(* Logix 5000 project; controller DC01 vendor 1 type 14 code 165 rev 32.12; software revision 32.04; part 2 of 13 *)
(* tags used below, declared in another part *)
   LN01_Main_Messages : DINT[250];
   LN01_Schedule : UDT_Current_Status;
   LN01_ScheduleUnits_Produced_from_line : DINT;
   LN01_Weekly_Schedule : UDT_Weekly_Schedule;

PROGRAM LN01   (* main routine MainRoutine *)
VAR
   Always_Off : BOOL;
   Average_Array : DINT[20] := ([0] := 1, [2] := 1, [8] := 1, [9] := 1);
   Average_Sum : DINT := 4;
   Averaged_LineSpeed : REAL := 0.0004;
   badModel : STRING_40;
   BlockStarveLocal : DINT;
   Break1_Hour : DINT;
   Break1_Hour_String : STRING;
   Break1_Length : DINT;
   Break1_MilliRemain : DINT;
   Break1_Min : DINT;
   Break1_Min_String : STRING;
   Break1_MinDisplay : DINT;
   Break1_SecDisplay : DINT;
   Break1_SecRemain : DINT;
   Break1_SecWholeMin : DINT;
   Break1_Timer : TIMER;
   Break2_Hour : DINT;
   Break2_Hour_String : STRING;
   Break2_Length : DINT;
   Break2_MilliRemain : DINT;
   Break2_Min : DINT;
   Break2_Min_String : STRING;
   Break2_MinDisplay : DINT;
   Break2_SecDisplay : DINT;
   Break2_SecRemain : DINT;
   Break2_SecWholeMin : DINT;
   Break2_Timer : TIMER;
   Break_1stStation : BOOL;
   Break_LineWide : BOOL;
   Break_WorkCenter : BOOL;
   Break_Workstation : BOOL;
   dlw_test : DINT := -805278210;
   End_Hour : DINT := 20;
   End_Hour_String : STRING := '20';
   End_Min : DINT := 3;
   End_Min_String : STRING := '3-';
   faultcount : DINT;
   FaultExists : CONTROL := (LEN := 230);
   firstCharacter : STRING_40 := 'W';
   FlexTimer_HoursDisplay : DINT;
   FlexTimer_MinutesDisplay : DINT;
   FlexTimer_SecondsDisplay : DINT;
   FlexTimertoHours : DINT;
   FlexTimertoMinutes : DINT;
   FlexTimertoSeconds : DINT;
   HoursFromMidnight : DINT;
   HoursFromMidnight_Remain : DINT;
   HoursTilMidnight : DINT;
   HoursTilMidnight_Remain : DINT;
   KnownFaultExist : DINT := 5;
   L02EAS35 : DINT;
   L02EDM16 : DINT;
   LineRate_perSecond_scheduled : DINT;
   LN01_Flex_Timer : TIMER;
   LN01_MachineOverAll_MNTa : DINT;
   LN01_MainLine_MSG : MESSAGE;
        MessageParameters(ServiceCode := 16#004c, LocalElement := LN01_Main_Messages[0], ...)
   LN01_ML_Message_MSG : MESSAGE;
   LN01_Rotate_Timer : TIMER;
   LN01_SNModel_MSG : MESSAGE;
   LN02EAS35 : DINT;
   LN02EDM16 : DINT;
   Local_Counter : COUNTER[20] := ([0].PRE := 1);
   Local_DATETIME : DINT[20];
   Local_Timer : TIMER[30] := ([0].EN := 1, [0].DN := 1, [3].PRE := 1000, [3].ACC := 429, [3].EN := 1, [3].TT := 1, [4].PRE := 400, [4].ACC := 272, [4].EN := 1, [4].TT := 1, [6].PRE := 2000, [6].ACC := 194, [6].EN := 1, [6].TT := 1);
   local_timer2 : TIMER := (PRE := 1000, ACC := 629, EN := 1, TT := 1);
   Lunch_Hour : DINT;
   Lunch_Hour_String : STRING;
   Lunch_Length : DINT;
   Lunch_MilliRemain : DINT;
   Lunch_Min : DINT;
   Lunch_Min_String : STRING;
   Lunch_MinDisplay : DINT;
   Lunch_SecDisplay : DINT;
   Lunch_SecRemain : DINT;
   Lunch_SecWholeMin : DINT;
   Lunch_Timer : TIMER;
   Midnight_Hour : DINT;
   mlc_test21 : BOOL;
   null : STRING;
   OneShot : DINT;
   ONS_0 : DINT := 536870912;
   ONS_20 : DINT;
   prevCalculateLocal : DINT;
   PreviousCount : DINT := 554;
   previousSerialNumber : STRING := 'CA0807422';
   PreviousShift : DINT := 1;
   readIndex : DINT := 41;
   register : DINT := 5;
   Rotate_MilliRemain : DINT;
   Rotate_Seconds_perShift : DINT;
   Rotate_SecRemain : DINT;
   RTO_Test : TIMER := (PRE := 2000, ACC := 2000, DN := 1);
   Scheduled_Units_Buffer : DINT := 1240;
   Shift_Break_Lengths : DINT;
   Shift_Break_Lengths_Remain : DINT;
   Shift_Delay_Min : DINT := 60;
   Shift_Extra_Min : DINT;
   Shift_Hours : DINT;
   Shift_Hours_Remain : DINT;
   Shift_Minutes : DINT;
   Shift_Minutes_Remain : DINT;
   Shift_Reset : BOOL;
   Shift_Reset_ONS : BOOL := 1;
   Shift_Seconds : DINT;
   Shift_Seconds_Remain : DINT;
   Start_Hour : DINT := 20;
   Start_Hour_String : STRING := '20';
   Start_Min : DINT := 3;
   Start_Min_String : STRING := '3-';
   tempIndex : DINT := 25;
   theoreticalUnitsReal : DINT;
   workstationid : DINT := 250;
   writeIndex : DINT := 42;
END_VAR

ROUTINE MainRoutine   (* ladder *)
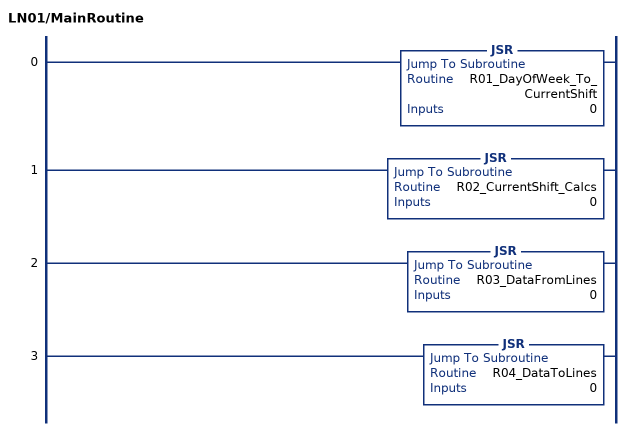
   0: JSR(R01_DayOfWeek_To_CurrentShift,0);
   1: JSR(R02_CurrentShift_Calcs,0);
   2: JSR(R03_DataFromLines,0);
   3: JSR(R04_DataToLines,0);
END_ROUTINE

ROUTINE R01_DayOfWeek_To_CurrentShift   (* ladder *)
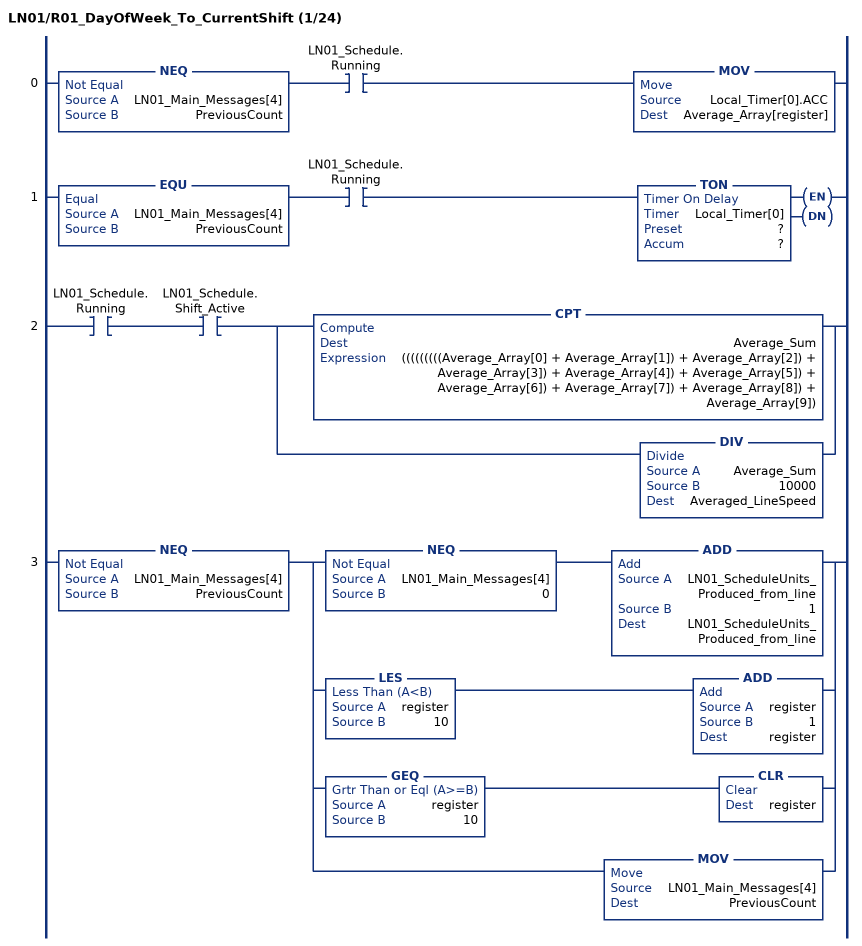
   0: NEQ(LN01_Main_Messages[4],PreviousCount)XIC(LN01_Schedule.Running)MOV(Local_Timer[0].ACC,Average_Array[register]);
   1: EQU(LN01_Main_Messages[4],PreviousCount)XIC(LN01_Schedule.Running)TON(Local_Timer[0],?,?);
   2: XIC(LN01_Schedule.Running)XIC(LN01_Schedule.Shift_Active)[CPT(Average_Sum,(((((((((Average_Array[0] + Average_Array[1]) + Average_Array[2]) + Average_Array[3]) + Average_Array[4]) + Average_Array[5]) + Average_Array[6]) + Average_Array[7]) + Average_Array[8]) + Average_Array[9])) ,DIV(Average_Sum,10000,Averaged_LineSpeed) ];
   3: NEQ(LN01_Main_Messages[4],PreviousCount)[NEQ(LN01_Main_Messages[4],0) ADD(LN01_ScheduleUnits_Produced_from_line,1,LN01_ScheduleUnits_Produced_from_line) ,LES(register,10) ADD(register,1,register) ,GEQ(register,10) CLR(register) ,MOV(LN01_Main_Messages[4],PreviousCount) ];
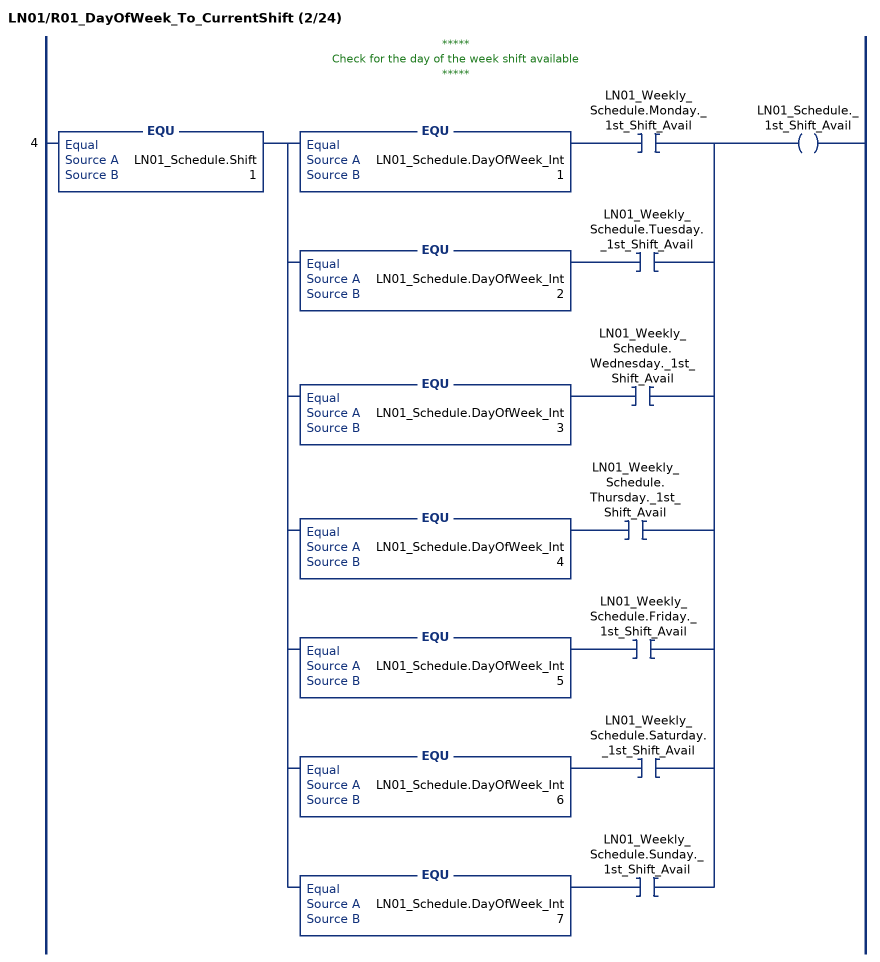
   // *****
   // Check for the day of the week shift available
   // *****
   4: EQU(LN01_Schedule.Shift,1)[EQU(LN01_Schedule.DayOfWeek_Int,1) XIC(LN01_Weekly_Schedule.Monday._1st_Shift_Avail) ,EQU(LN01_Schedule.DayOfWeek_Int,2) XIC(LN01_Weekly_Schedule.Tuesday._1st_Shift_Avail) ,EQU(LN01_Schedule.DayOfWeek_Int,3) XIC(LN01_Weekly_Schedule.Wednesday._1st_Shift_Avail) ,EQU(LN01_Schedule.DayOfWeek_Int,4) XIC(LN01_Weekly_Schedule.Thursday._1st_Shift_Avail) ,EQU(LN01_Schedule.DayOfWeek_Int,5) XIC(LN01_Weekly_Schedule.Friday._1st_Shift_Avail) ,EQU(LN01_Schedule.DayOfWeek_Int,6) XIC(LN01_Weekly_Schedule.Saturday._1st_Shift_Avail) ,EQU(LN01_Schedule.DayOfWeek_Int,7) XIC(LN01_Weekly_Schedule.Sunday._1st_Shift_Avail) ]OTE(LN01_Schedule._1st_Shift_Avail);
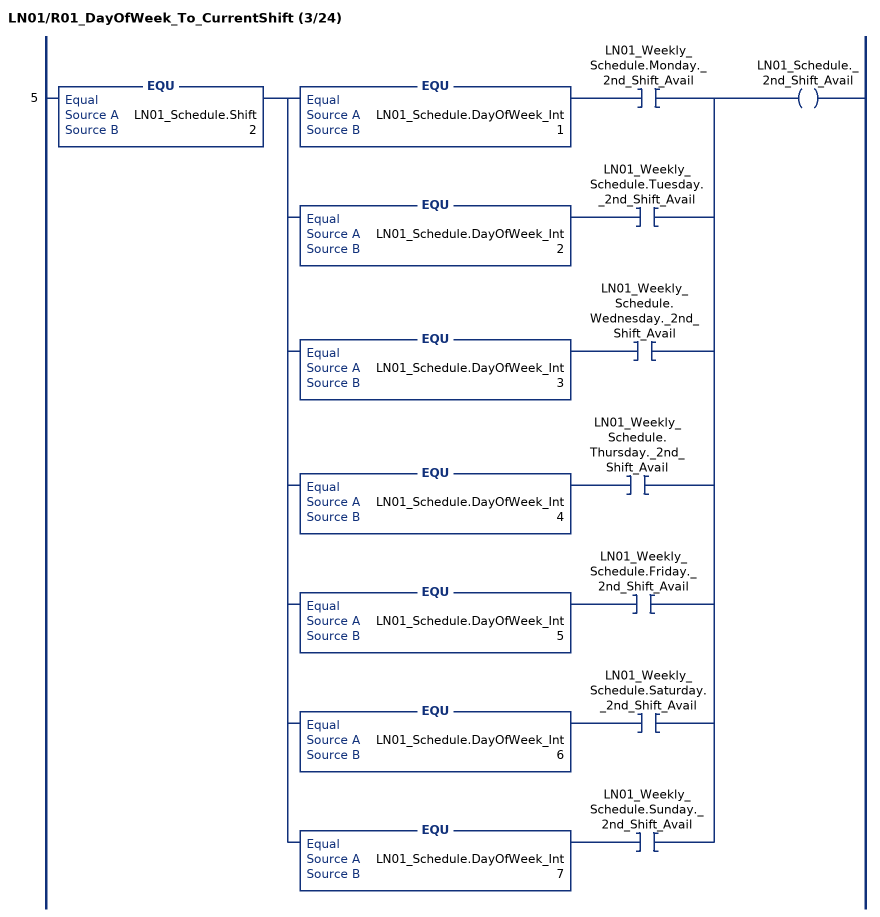
   5: EQU(LN01_Schedule.Shift,2)[EQU(LN01_Schedule.DayOfWeek_Int,1) XIC(LN01_Weekly_Schedule.Monday._2nd_Shift_Avail) ,EQU(LN01_Schedule.DayOfWeek_Int,2) XIC(LN01_Weekly_Schedule.Tuesday._2nd_Shift_Avail) ,EQU(LN01_Schedule.DayOfWeek_Int,3) XIC(LN01_Weekly_Schedule.Wednesday._2nd_Shift_Avail) ,EQU(LN01_Schedule.DayOfWeek_Int,4) XIC(LN01_Weekly_Schedule.Thursday._2nd_Shift_Avail) ,EQU(LN01_Schedule.DayOfWeek_Int,5) XIC(LN01_Weekly_Schedule.Friday._2nd_Shift_Avail) ,EQU(LN01_Schedule.DayOfWeek_Int,6) XIC(LN01_Weekly_Schedule.Saturday._2nd_Shift_Avail) ,EQU(LN01_Schedule.DayOfWeek_Int,7) XIC(LN01_Weekly_Schedule.Sunday._2nd_Shift_Avail) ]OTE(LN01_Schedule._2nd_Shift_Avail);
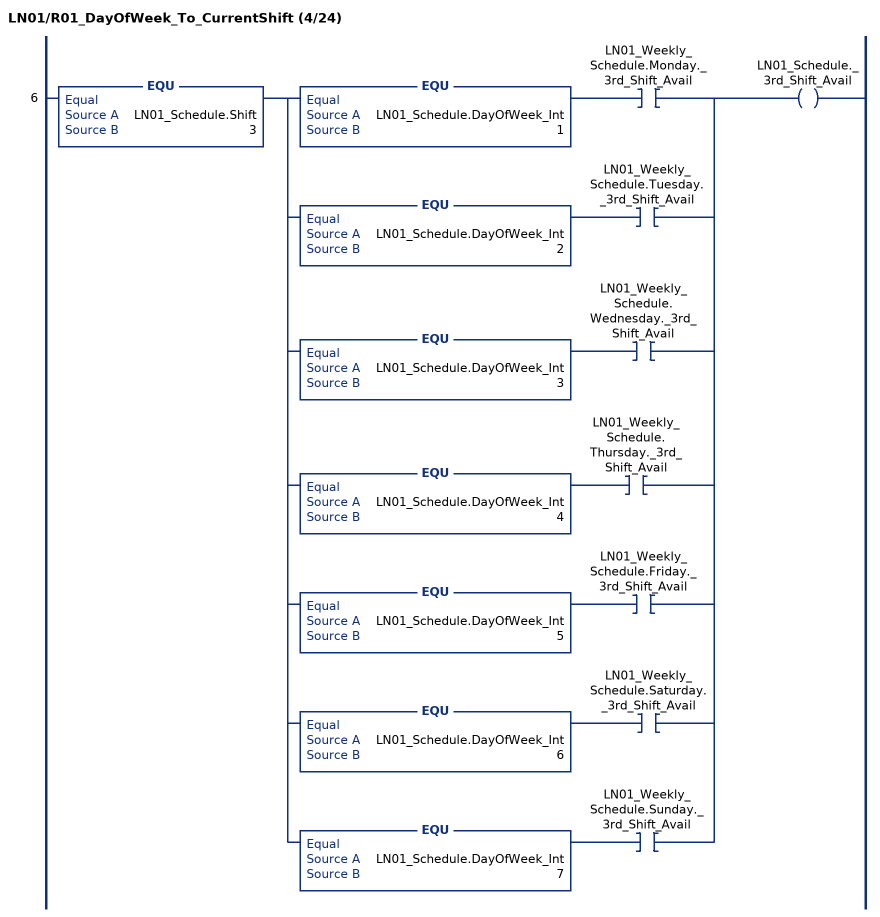
   6: EQU(LN01_Schedule.Shift,3)[EQU(LN01_Schedule.DayOfWeek_Int,1) XIC(LN01_Weekly_Schedule.Monday._3rd_Shift_Avail) ,EQU(LN01_Schedule.DayOfWeek_Int,2) XIC(LN01_Weekly_Schedule.Tuesday._3rd_Shift_Avail) ,EQU(LN01_Schedule.DayOfWeek_Int,3) XIC(LN01_Weekly_Schedule.Wednesday._3rd_Shift_Avail) ,EQU(LN01_Schedule.DayOfWeek_Int,4) XIC(LN01_Weekly_Schedule.Thursday._3rd_Shift_Avail) ,EQU(LN01_Schedule.DayOfWeek_Int,5) XIC(LN01_Weekly_Schedule.Friday._3rd_Shift_Avail) ,EQU(LN01_Schedule.DayOfWeek_Int,6) XIC(LN01_Weekly_Schedule.Saturday._3rd_Shift_Avail) ,EQU(LN01_Schedule.DayOfWeek_Int,7) XIC(LN01_Weekly_Schedule.Sunday._3rd_Shift_Avail) ]OTE(LN01_Schedule._3rd_Shift_Avail);
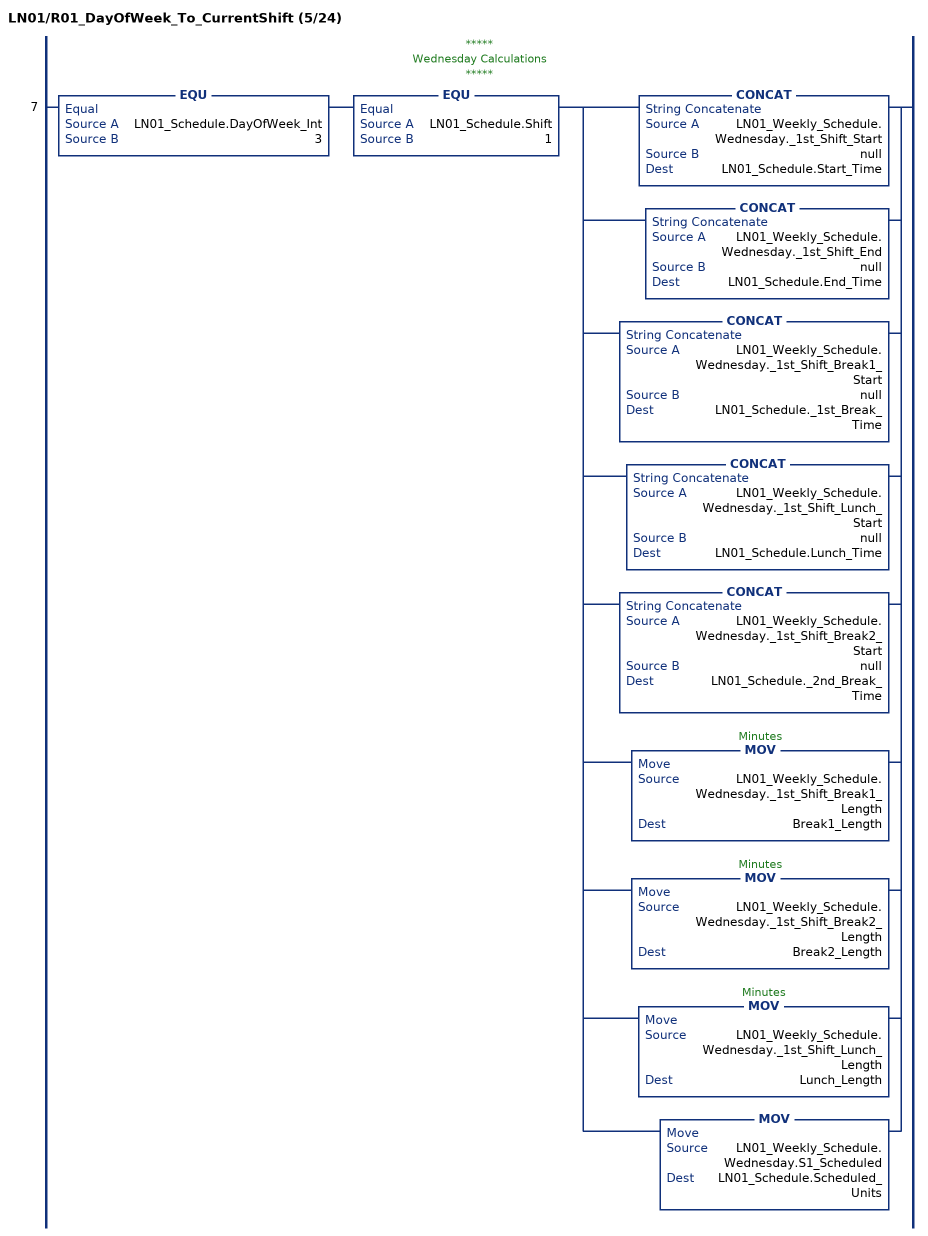
   // *****
   // Wednesday Calculations
   // *****
   7: EQU(LN01_Schedule.DayOfWeek_Int,3)EQU(LN01_Schedule.Shift,1)[CONCAT(LN01_Weekly_Schedule.Wednesday._1st_Shift_Start,null,LN01_Schedule.Start_Time) ,CONCAT(LN01_Weekly_Schedule.Wednesday._1st_Shift_End,null,LN01_Schedule.End_Time) ,CONCAT(LN01_Weekly_Schedule.Wednesday._1st_Shift_Break1_Start,null,LN01_Schedule._1st_Break_Time) ,CONCAT(LN01_Weekly_Schedule.Wednesday._1st_Shift_Lunch_Start,null,LN01_Schedule.Lunch_Time) ,CONCAT(LN01_Weekly_Schedule.Wednesday._1st_Shift_Break2_Start,null,LN01_Schedule._2nd_Break_Time) ,MOV(LN01_Weekly_Schedule.Wednesday._1st_Shift_Break1_Length,Break1_Length) ,MOV(LN01_Weekly_Schedule.Wednesday._1st_Shift_Break2_Length,Break2_Length) ,MOV(LN01_Weekly_Schedule.Wednesday._1st_Shift_Lunch_Length,Lunch_Length) ,MOV(LN01_Weekly_Schedule.Wednesday.S1_Scheduled,LN01_Schedule.Scheduled_Units) ];
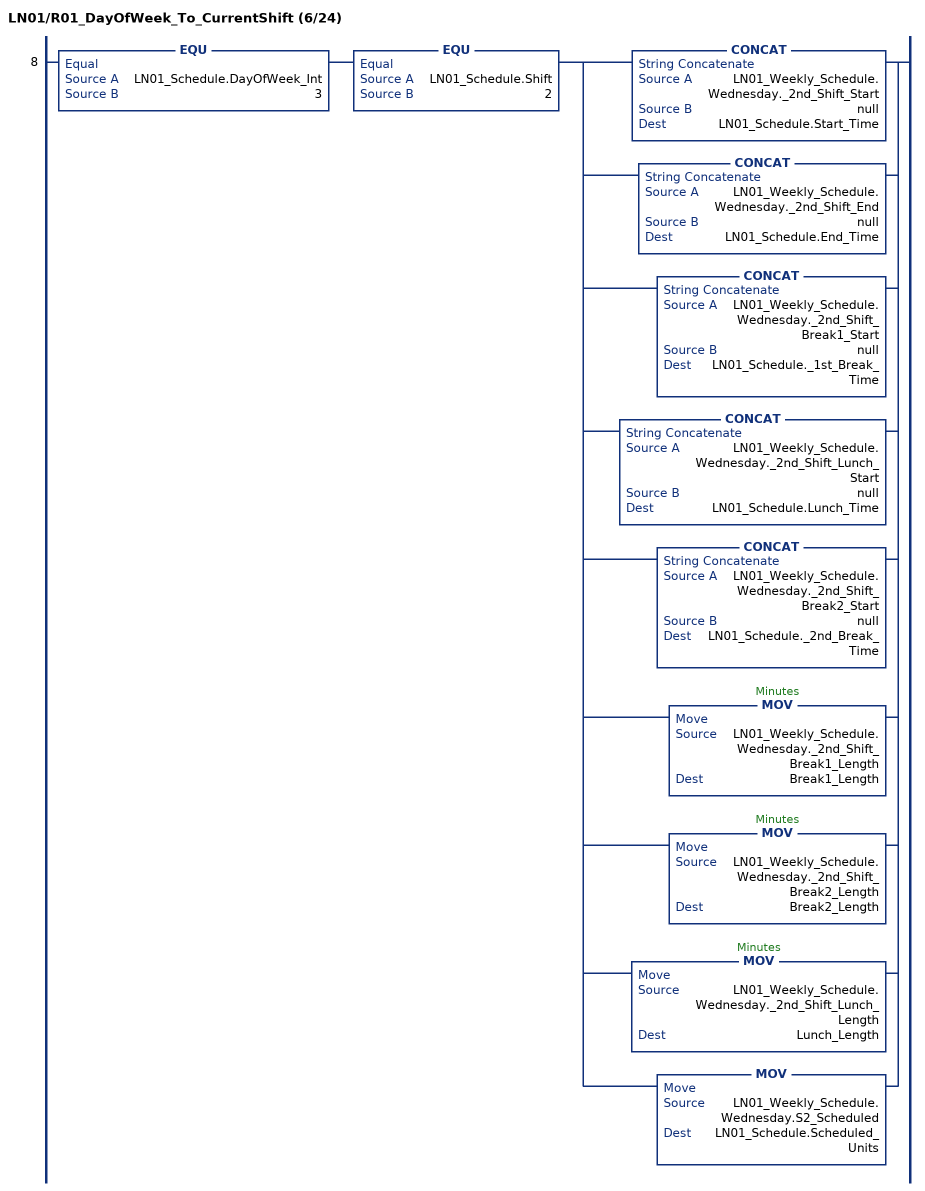
   8: EQU(LN01_Schedule.DayOfWeek_Int,3)EQU(LN01_Schedule.Shift,2)[CONCAT(LN01_Weekly_Schedule.Wednesday._2nd_Shift_Start,null,LN01_Schedule.Start_Time) ,CONCAT(LN01_Weekly_Schedule.Wednesday._2nd_Shift_End,null,LN01_Schedule.End_Time) ,CONCAT(LN01_Weekly_Schedule.Wednesday._2nd_Shift_Break1_Start,null,LN01_Schedule._1st_Break_Time) ,CONCAT(LN01_Weekly_Schedule.Wednesday._2nd_Shift_Lunch_Start,null,LN01_Schedule.Lunch_Time) ,CONCAT(LN01_Weekly_Schedule.Wednesday._2nd_Shift_Break2_Start,null,LN01_Schedule._2nd_Break_Time) ,MOV(LN01_Weekly_Schedule.Wednesday._2nd_Shift_Break1_Length,Break1_Length) ,MOV(LN01_Weekly_Schedule.Wednesday._2nd_Shift_Break2_Length,Break2_Length) ,MOV(LN01_Weekly_Schedule.Wednesday._2nd_Shift_Lunch_Length,Lunch_Length) ,MOV(LN01_Weekly_Schedule.Wednesday.S2_Scheduled,LN01_Schedule.Scheduled_Units) ];
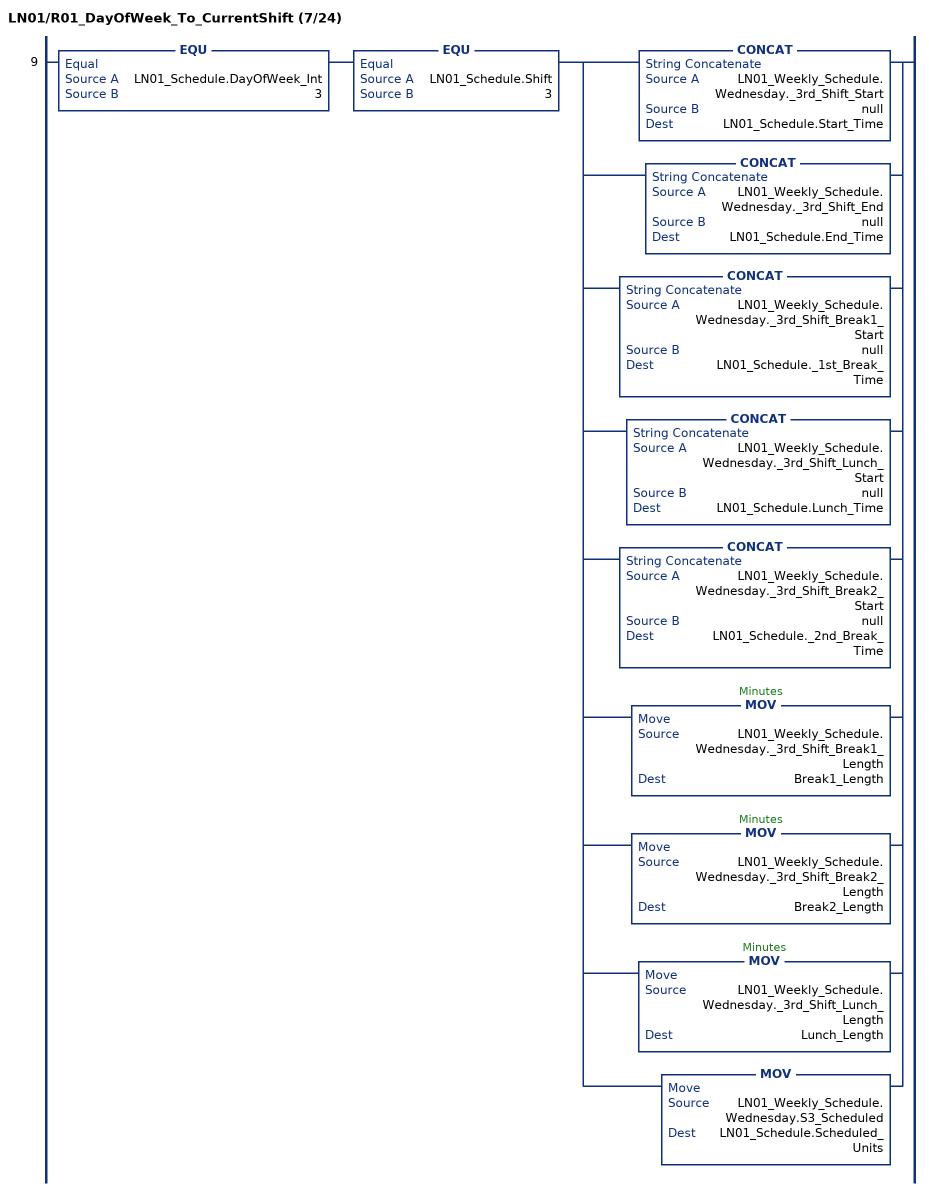
   9: EQU(LN01_Schedule.DayOfWeek_Int,3)EQU(LN01_Schedule.Shift,3)[CONCAT(LN01_Weekly_Schedule.Wednesday._3rd_Shift_Start,null,LN01_Schedule.Start_Time) ,CONCAT(LN01_Weekly_Schedule.Wednesday._3rd_Shift_End,null,LN01_Schedule.End_Time) ,CONCAT(LN01_Weekly_Schedule.Wednesday._3rd_Shift_Break1_Start,null,LN01_Schedule._1st_Break_Time) ,CONCAT(LN01_Weekly_Schedule.Wednesday._3rd_Shift_Lunch_Start,null,LN01_Schedule.Lunch_Time) ,CONCAT(LN01_Weekly_Schedule.Wednesday._3rd_Shift_Break2_Start,null,LN01_Schedule._2nd_Break_Time) ,MOV(LN01_Weekly_Schedule.Wednesday._3rd_Shift_Break1_Length,Break1_Length) ,MOV(LN01_Weekly_Schedule.Wednesday._3rd_Shift_Break2_Length,Break2_Length) ,MOV(LN01_Weekly_Schedule.Wednesday._3rd_Shift_Lunch_Length,Lunch_Length) ,MOV(LN01_Weekly_Schedule.Wednesday.S3_Scheduled,LN01_Schedule.Scheduled_Units) ];
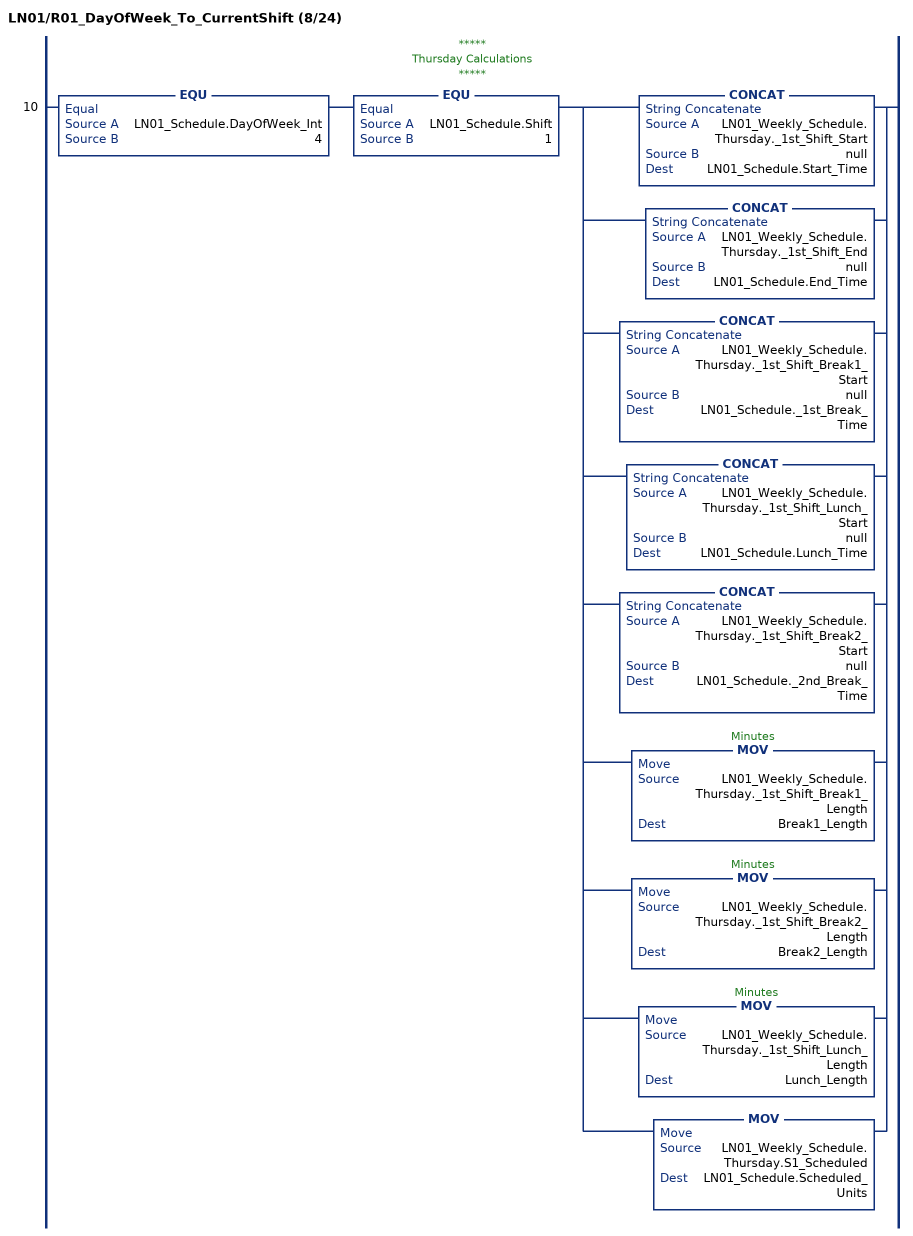
   // *****
   // Thursday Calculations
   // *****
   10: EQU(LN01_Schedule.DayOfWeek_Int,4)EQU(LN01_Schedule.Shift,1)[CONCAT(LN01_Weekly_Schedule.Thursday._1st_Shift_Start,null,LN01_Schedule.Start_Time) ,CONCAT(LN01_Weekly_Schedule.Thursday._1st_Shift_End,null,LN01_Schedule.End_Time) ,CONCAT(LN01_Weekly_Schedule.Thursday._1st_Shift_Break1_Start,null,LN01_Schedule._1st_Break_Time) ,CONCAT(LN01_Weekly_Schedule.Thursday._1st_Shift_Lunch_Start,null,LN01_Schedule.Lunch_Time) ,CONCAT(LN01_Weekly_Schedule.Thursday._1st_Shift_Break2_Start,null,LN01_Schedule._2nd_Break_Time) ,MOV(LN01_Weekly_Schedule.Thursday._1st_Shift_Break1_Length,Break1_Length) ,MOV(LN01_Weekly_Schedule.Thursday._1st_Shift_Break2_Length,Break2_Length) ,MOV(LN01_Weekly_Schedule.Thursday._1st_Shift_Lunch_Length,Lunch_Length) ,MOV(LN01_Weekly_Schedule.Thursday.S1_Scheduled,LN01_Schedule.Scheduled_Units) ];
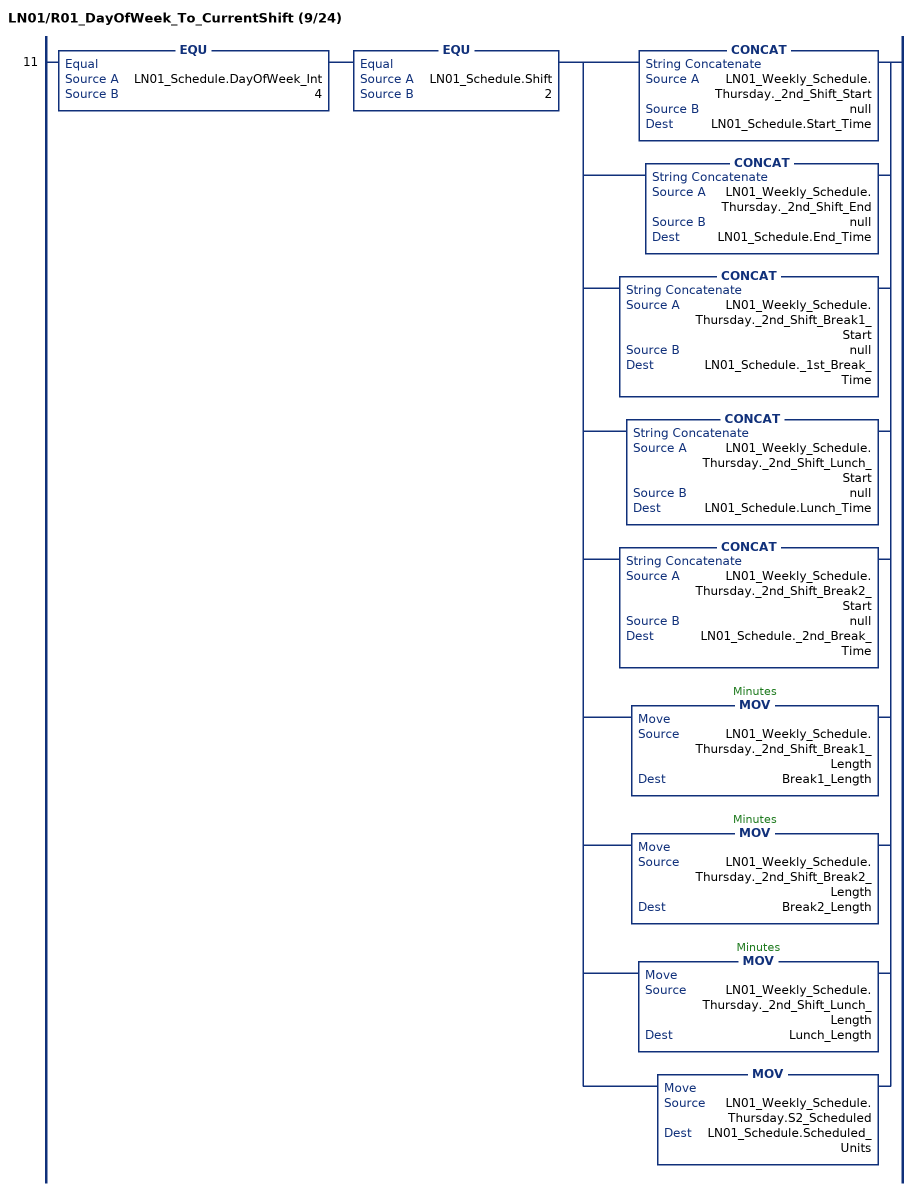
   11: EQU(LN01_Schedule.DayOfWeek_Int,4)EQU(LN01_Schedule.Shift,2)[CONCAT(LN01_Weekly_Schedule.Thursday._2nd_Shift_Start,null,LN01_Schedule.Start_Time) ,CONCAT(LN01_Weekly_Schedule.Thursday._2nd_Shift_End,null,LN01_Schedule.End_Time) ,CONCAT(LN01_Weekly_Schedule.Thursday._2nd_Shift_Break1_Start,null,LN01_Schedule._1st_Break_Time) ,CONCAT(LN01_Weekly_Schedule.Thursday._2nd_Shift_Lunch_Start,null,LN01_Schedule.Lunch_Time) ,CONCAT(LN01_Weekly_Schedule.Thursday._2nd_Shift_Break2_Start,null,LN01_Schedule._2nd_Break_Time) ,MOV(LN01_Weekly_Schedule.Thursday._2nd_Shift_Break1_Length,Break1_Length) ,MOV(LN01_Weekly_Schedule.Thursday._2nd_Shift_Break2_Length,Break2_Length) ,MOV(LN01_Weekly_Schedule.Thursday._2nd_Shift_Lunch_Length,Lunch_Length) ,MOV(LN01_Weekly_Schedule.Thursday.S2_Scheduled,LN01_Schedule.Scheduled_Units) ];
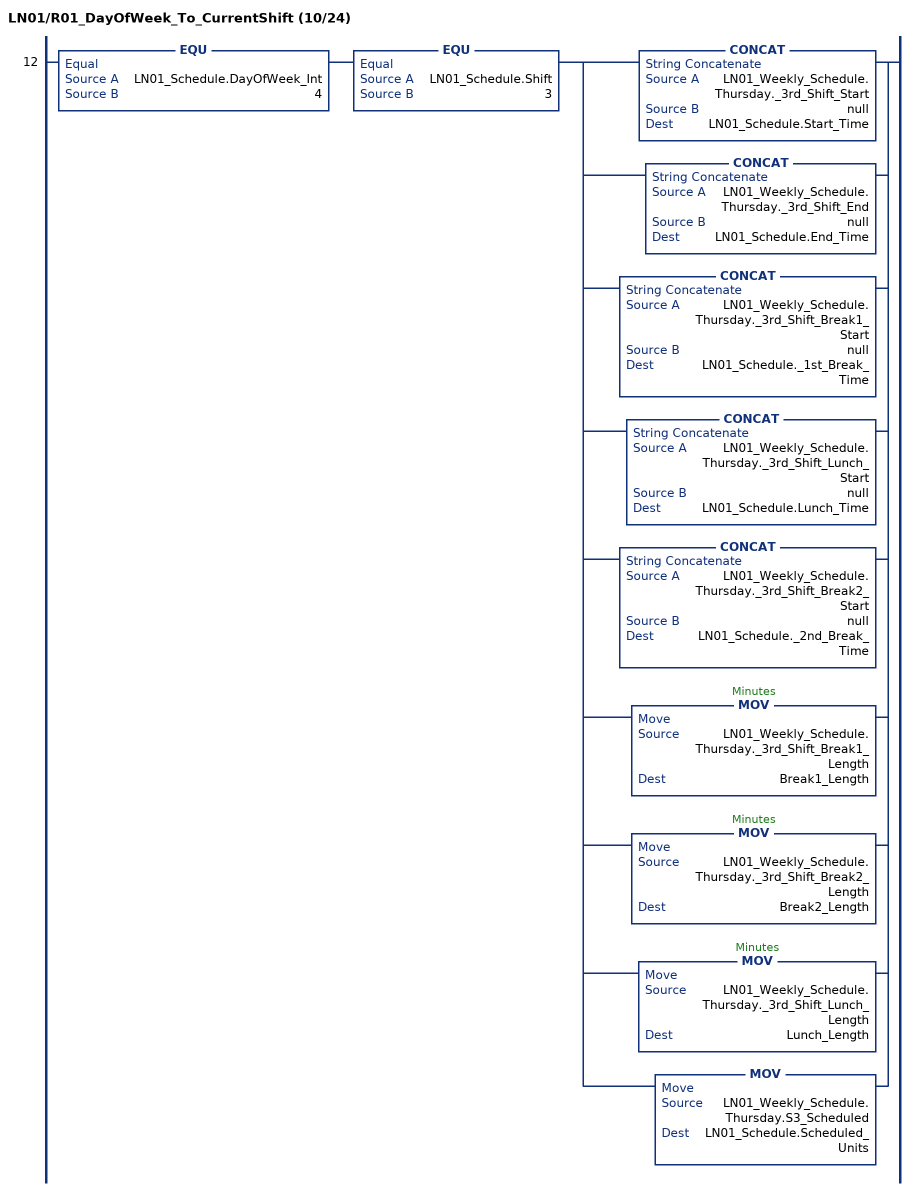
   12: EQU(LN01_Schedule.DayOfWeek_Int,4)EQU(LN01_Schedule.Shift,3)[CONCAT(LN01_Weekly_Schedule.Thursday._3rd_Shift_Start,null,LN01_Schedule.Start_Time) ,CONCAT(LN01_Weekly_Schedule.Thursday._3rd_Shift_End,null,LN01_Schedule.End_Time) ,CONCAT(LN01_Weekly_Schedule.Thursday._3rd_Shift_Break1_Start,null,LN01_Schedule._1st_Break_Time) ,CONCAT(LN01_Weekly_Schedule.Thursday._3rd_Shift_Lunch_Start,null,LN01_Schedule.Lunch_Time) ,CONCAT(LN01_Weekly_Schedule.Thursday._3rd_Shift_Break2_Start,null,LN01_Schedule._2nd_Break_Time) ,MOV(LN01_Weekly_Schedule.Thursday._3rd_Shift_Break1_Length,Break1_Length) ,MOV(LN01_Weekly_Schedule.Thursday._3rd_Shift_Break2_Length,Break2_Length) ,MOV(LN01_Weekly_Schedule.Thursday._3rd_Shift_Lunch_Length,Lunch_Length) ,MOV(LN01_Weekly_Schedule.Thursday.S3_Scheduled,LN01_Schedule.Scheduled_Units) ];
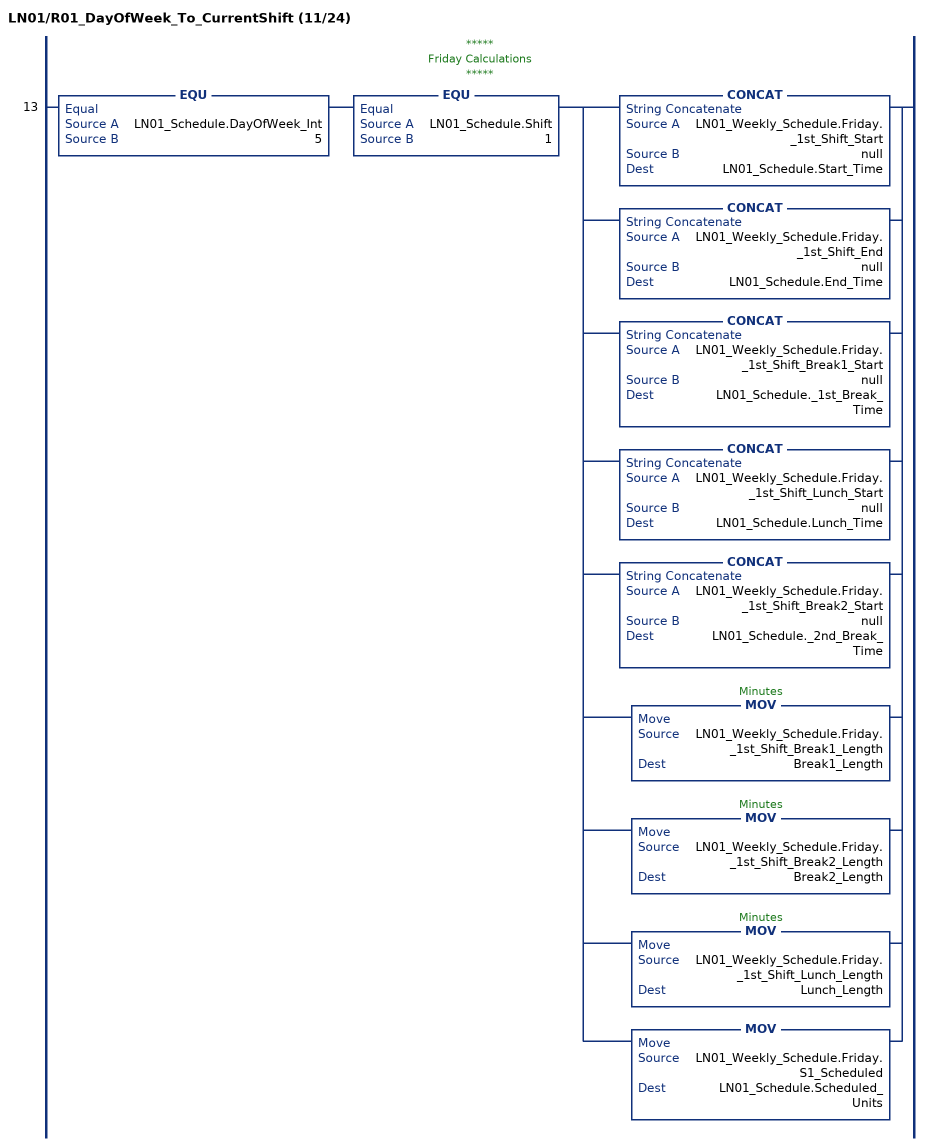
   // *****
   // Friday Calculations
   // *****
   13: EQU(LN01_Schedule.DayOfWeek_Int,5)EQU(LN01_Schedule.Shift,1)[CONCAT(LN01_Weekly_Schedule.Friday._1st_Shift_Start,null,LN01_Schedule.Start_Time) ,CONCAT(LN01_Weekly_Schedule.Friday._1st_Shift_End,null,LN01_Schedule.End_Time) ,CONCAT(LN01_Weekly_Schedule.Friday._1st_Shift_Break1_Start,null,LN01_Schedule._1st_Break_Time) ,CONCAT(LN01_Weekly_Schedule.Friday._1st_Shift_Lunch_Start,null,LN01_Schedule.Lunch_Time) ,CONCAT(LN01_Weekly_Schedule.Friday._1st_Shift_Break2_Start,null,LN01_Schedule._2nd_Break_Time) ,MOV(LN01_Weekly_Schedule.Friday._1st_Shift_Break1_Length,Break1_Length) ,MOV(LN01_Weekly_Schedule.Friday._1st_Shift_Break2_Length,Break2_Length) ,MOV(LN01_Weekly_Schedule.Friday._1st_Shift_Lunch_Length,Lunch_Length) ,MOV(LN01_Weekly_Schedule.Friday.S1_Scheduled,LN01_Schedule.Scheduled_Units) ];
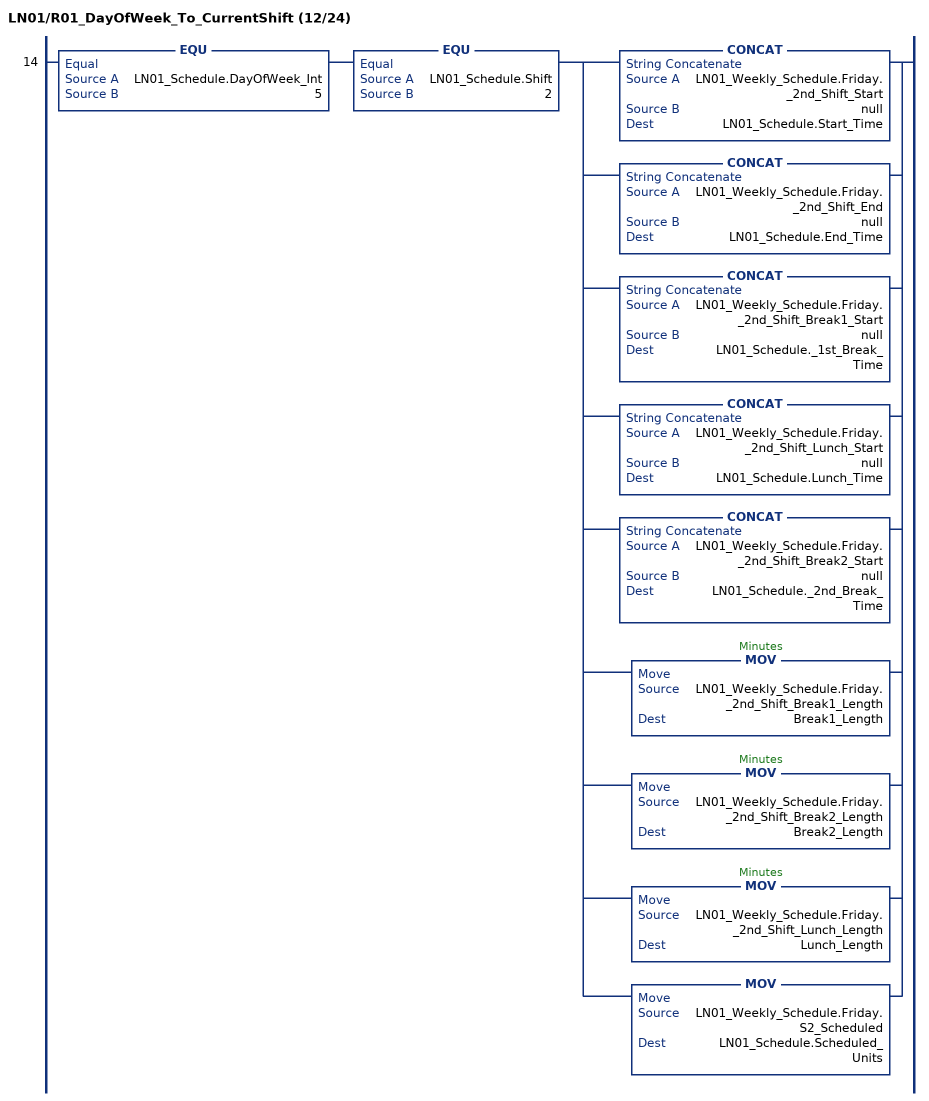
   14: EQU(LN01_Schedule.DayOfWeek_Int,5)EQU(LN01_Schedule.Shift,2)[CONCAT(LN01_Weekly_Schedule.Friday._2nd_Shift_Start,null,LN01_Schedule.Start_Time) ,CONCAT(LN01_Weekly_Schedule.Friday._2nd_Shift_End,null,LN01_Schedule.End_Time) ,CONCAT(LN01_Weekly_Schedule.Friday._2nd_Shift_Break1_Start,null,LN01_Schedule._1st_Break_Time) ,CONCAT(LN01_Weekly_Schedule.Friday._2nd_Shift_Lunch_Start,null,LN01_Schedule.Lunch_Time) ,CONCAT(LN01_Weekly_Schedule.Friday._2nd_Shift_Break2_Start,null,LN01_Schedule._2nd_Break_Time) ,MOV(LN01_Weekly_Schedule.Friday._2nd_Shift_Break1_Length,Break1_Length) ,MOV(LN01_Weekly_Schedule.Friday._2nd_Shift_Break2_Length,Break2_Length) ,MOV(LN01_Weekly_Schedule.Friday._2nd_Shift_Lunch_Length,Lunch_Length) ,MOV(LN01_Weekly_Schedule.Friday.S2_Scheduled,LN01_Schedule.Scheduled_Units) ];
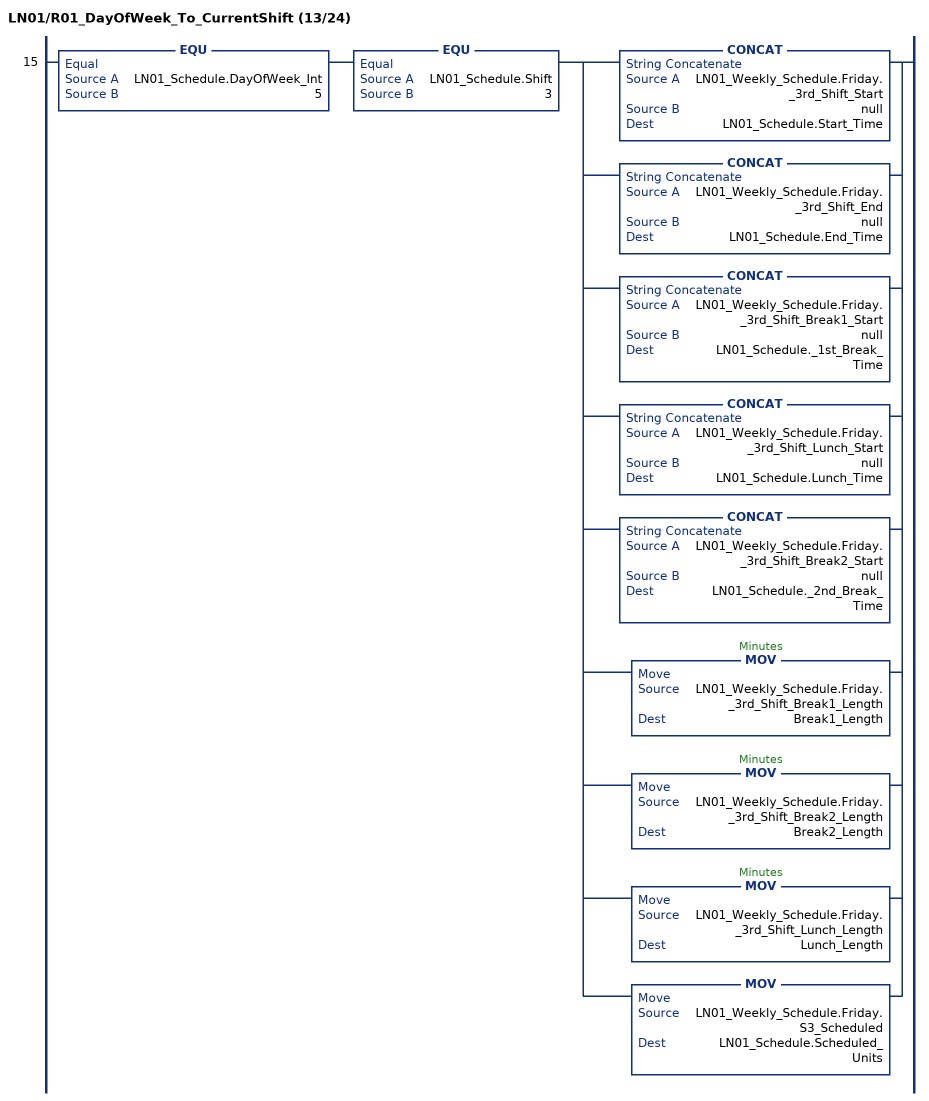
   15: EQU(LN01_Schedule.DayOfWeek_Int,5)EQU(LN01_Schedule.Shift,3)[CONCAT(LN01_Weekly_Schedule.Friday._3rd_Shift_Start,null,LN01_Schedule.Start_Time) ,CONCAT(LN01_Weekly_Schedule.Friday._3rd_Shift_End,null,LN01_Schedule.End_Time) ,CONCAT(LN01_Weekly_Schedule.Friday._3rd_Shift_Break1_Start,null,LN01_Schedule._1st_Break_Time) ,CONCAT(LN01_Weekly_Schedule.Friday._3rd_Shift_Lunch_Start,null,LN01_Schedule.Lunch_Time) ,CONCAT(LN01_Weekly_Schedule.Friday._3rd_Shift_Break2_Start,null,LN01_Schedule._2nd_Break_Time) ,MOV(LN01_Weekly_Schedule.Friday._3rd_Shift_Break1_Length,Break1_Length) ,MOV(LN01_Weekly_Schedule.Friday._3rd_Shift_Break2_Length,Break2_Length) ,MOV(LN01_Weekly_Schedule.Friday._3rd_Shift_Lunch_Length,Lunch_Length) ,MOV(LN01_Weekly_Schedule.Friday.S3_Scheduled,LN01_Schedule.Scheduled_Units) ];
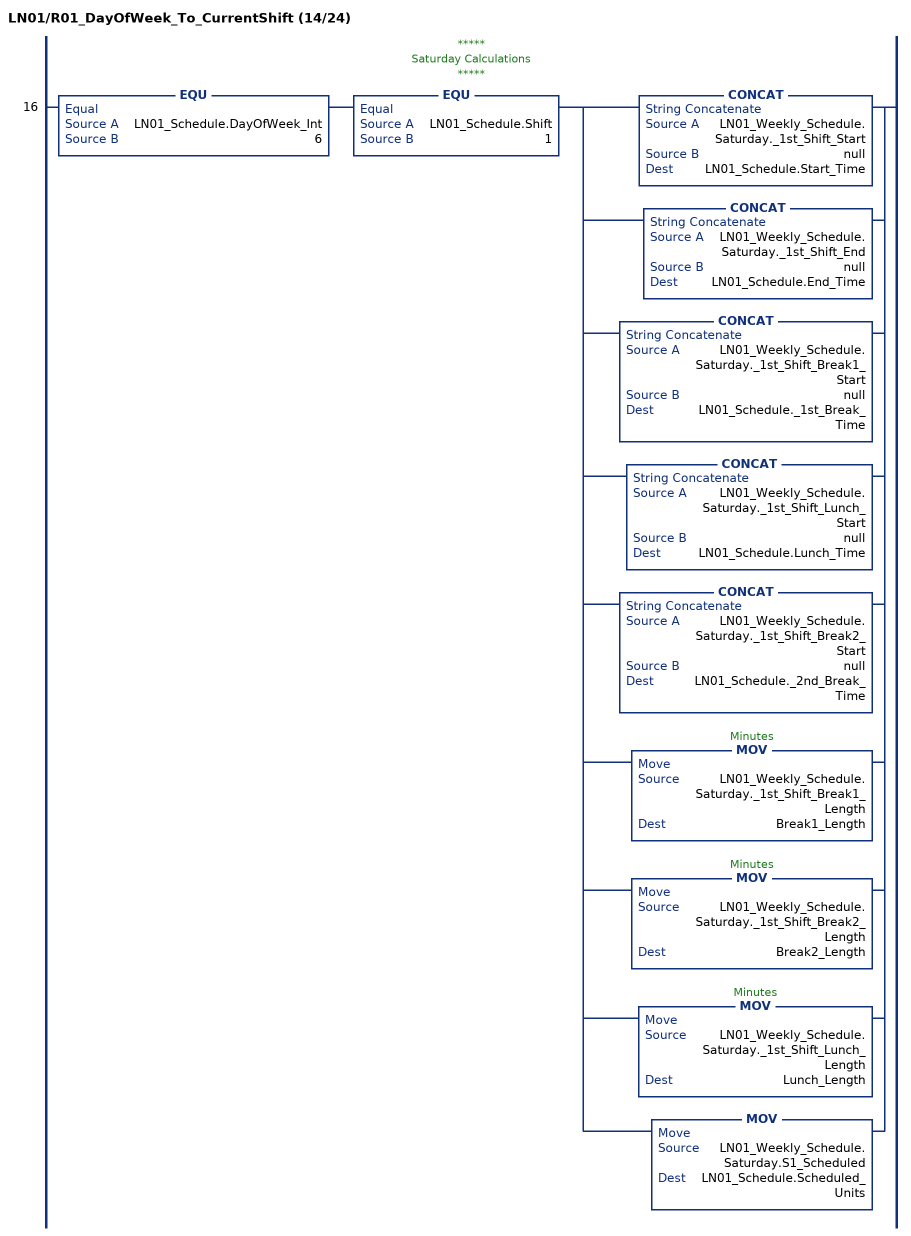
   // *****
   // Saturday Calculations
   // *****
   16: EQU(LN01_Schedule.DayOfWeek_Int,6)EQU(LN01_Schedule.Shift,1)[CONCAT(LN01_Weekly_Schedule.Saturday._1st_Shift_Start,null,LN01_Schedule.Start_Time) ,CONCAT(LN01_Weekly_Schedule.Saturday._1st_Shift_End,null,LN01_Schedule.End_Time) ,CONCAT(LN01_Weekly_Schedule.Saturday._1st_Shift_Break1_Start,null,LN01_Schedule._1st_Break_Time) ,CONCAT(LN01_Weekly_Schedule.Saturday._1st_Shift_Lunch_Start,null,LN01_Schedule.Lunch_Time) ,CONCAT(LN01_Weekly_Schedule.Saturday._1st_Shift_Break2_Start,null,LN01_Schedule._2nd_Break_Time) ,MOV(LN01_Weekly_Schedule.Saturday._1st_Shift_Break1_Length,Break1_Length) ,MOV(LN01_Weekly_Schedule.Saturday._1st_Shift_Break2_Length,Break2_Length) ,MOV(LN01_Weekly_Schedule.Saturday._1st_Shift_Lunch_Length,Lunch_Length) ,MOV(LN01_Weekly_Schedule.Saturday.S1_Scheduled,LN01_Schedule.Scheduled_Units) ];
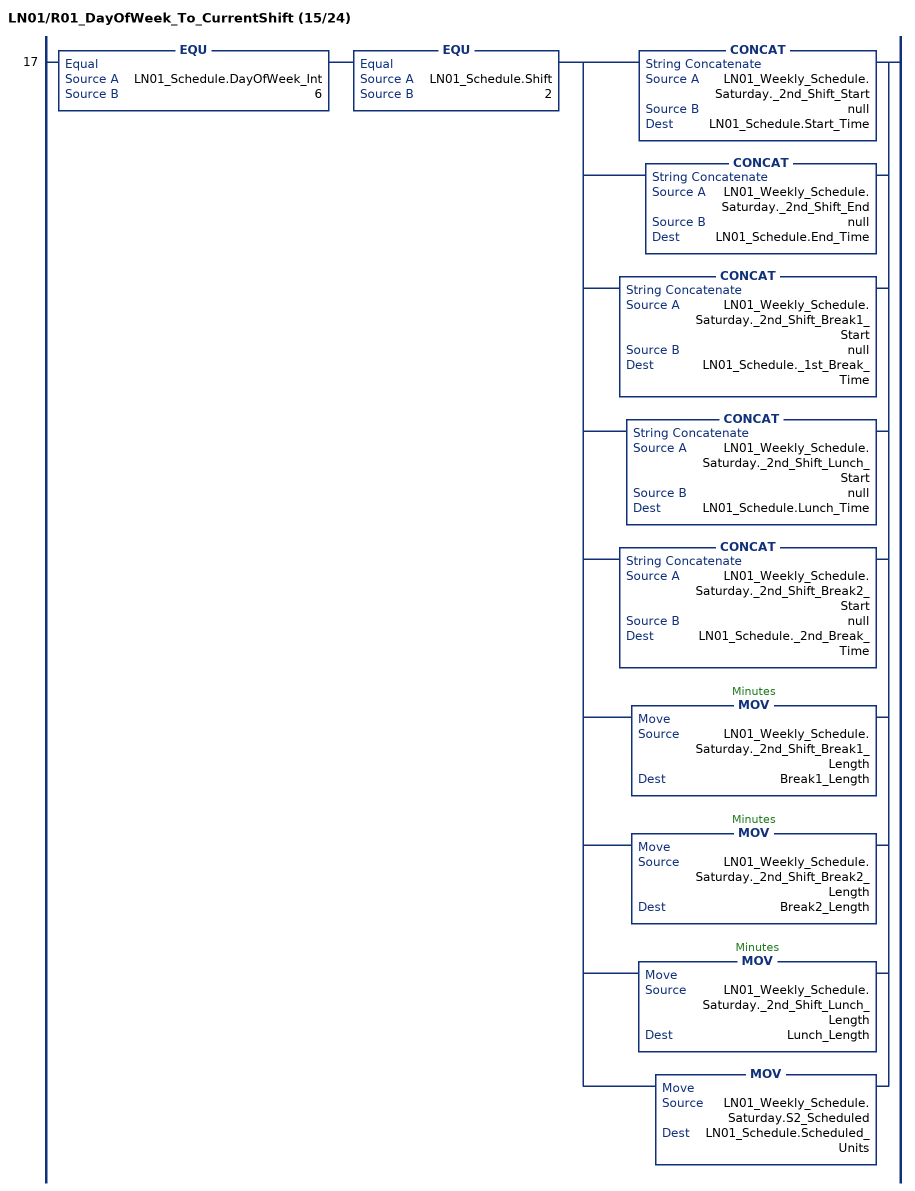
   17: EQU(LN01_Schedule.DayOfWeek_Int,6)EQU(LN01_Schedule.Shift,2)[CONCAT(LN01_Weekly_Schedule.Saturday._2nd_Shift_Start,null,LN01_Schedule.Start_Time) ,CONCAT(LN01_Weekly_Schedule.Saturday._2nd_Shift_End,null,LN01_Schedule.End_Time) ,CONCAT(LN01_Weekly_Schedule.Saturday._2nd_Shift_Break1_Start,null,LN01_Schedule._1st_Break_Time) ,CONCAT(LN01_Weekly_Schedule.Saturday._2nd_Shift_Lunch_Start,null,LN01_Schedule.Lunch_Time) ,CONCAT(LN01_Weekly_Schedule.Saturday._2nd_Shift_Break2_Start,null,LN01_Schedule._2nd_Break_Time) ,MOV(LN01_Weekly_Schedule.Saturday._2nd_Shift_Break1_Length,Break1_Length) ,MOV(LN01_Weekly_Schedule.Saturday._2nd_Shift_Break2_Length,Break2_Length) ,MOV(LN01_Weekly_Schedule.Saturday._2nd_Shift_Lunch_Length,Lunch_Length) ,MOV(LN01_Weekly_Schedule.Saturday.S2_Scheduled,LN01_Schedule.Scheduled_Units) ];
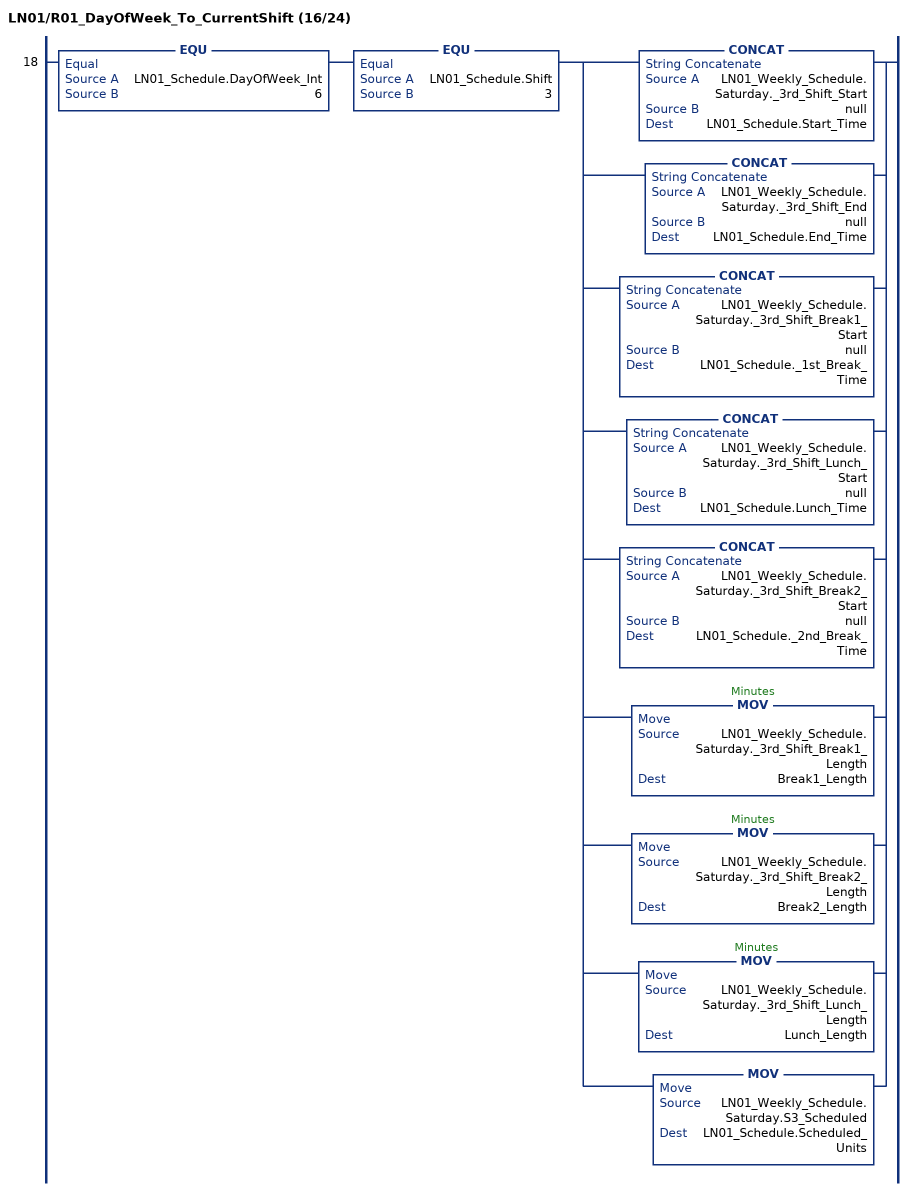
   18: EQU(LN01_Schedule.DayOfWeek_Int,6)EQU(LN01_Schedule.Shift,3)[CONCAT(LN01_Weekly_Schedule.Saturday._3rd_Shift_Start,null,LN01_Schedule.Start_Time) ,CONCAT(LN01_Weekly_Schedule.Saturday._3rd_Shift_End,null,LN01_Schedule.End_Time) ,CONCAT(LN01_Weekly_Schedule.Saturday._3rd_Shift_Break1_Start,null,LN01_Schedule._1st_Break_Time) ,CONCAT(LN01_Weekly_Schedule.Saturday._3rd_Shift_Lunch_Start,null,LN01_Schedule.Lunch_Time) ,CONCAT(LN01_Weekly_Schedule.Saturday._3rd_Shift_Break2_Start,null,LN01_Schedule._2nd_Break_Time) ,MOV(LN01_Weekly_Schedule.Saturday._3rd_Shift_Break1_Length,Break1_Length) ,MOV(LN01_Weekly_Schedule.Saturday._3rd_Shift_Break2_Length,Break2_Length) ,MOV(LN01_Weekly_Schedule.Saturday._3rd_Shift_Lunch_Length,Lunch_Length) ,MOV(LN01_Weekly_Schedule.Saturday.S3_Scheduled,LN01_Schedule.Scheduled_Units) ];
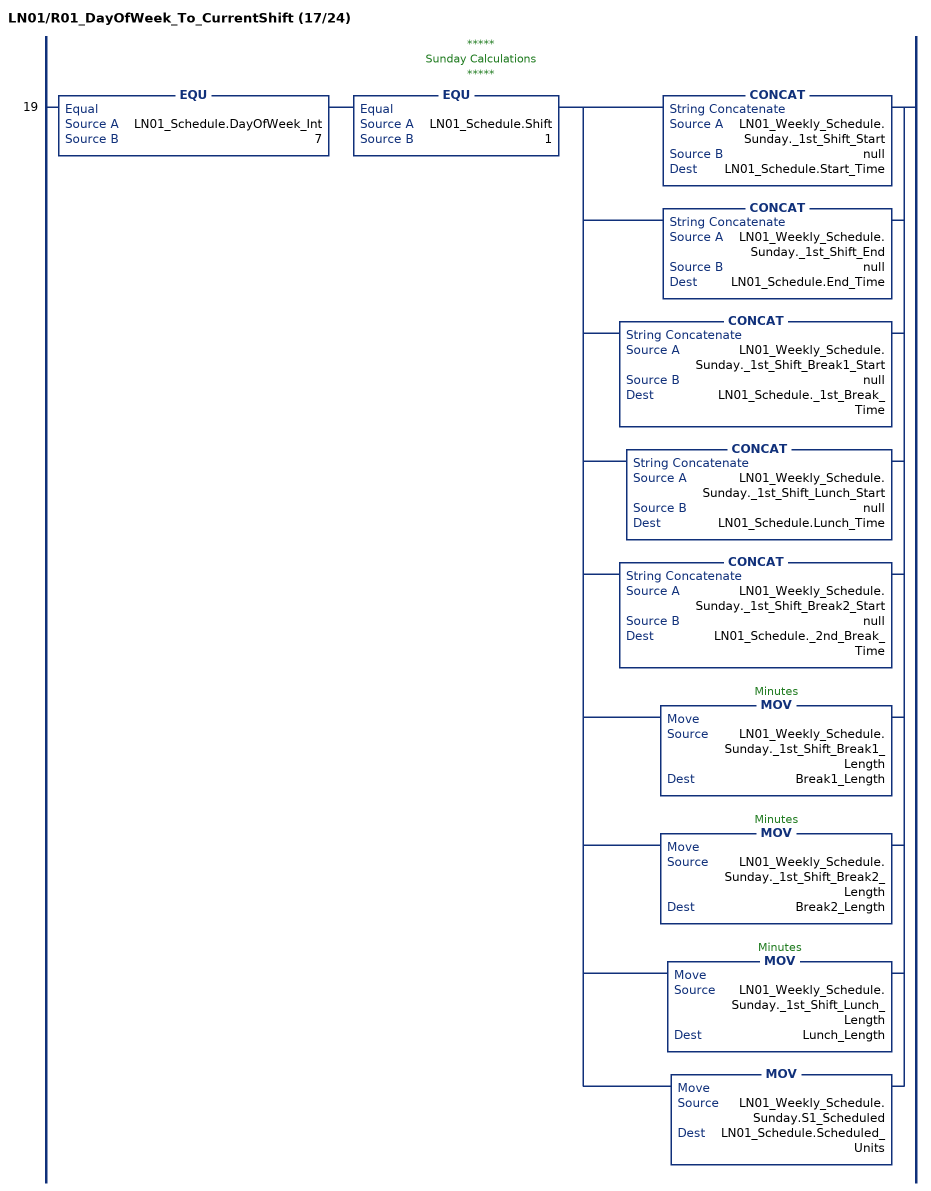
   // *****
   // Sunday Calculations
   // *****
   19: EQU(LN01_Schedule.DayOfWeek_Int,7)EQU(LN01_Schedule.Shift,1)[CONCAT(LN01_Weekly_Schedule.Sunday._1st_Shift_Start,null,LN01_Schedule.Start_Time) ,CONCAT(LN01_Weekly_Schedule.Sunday._1st_Shift_End,null,LN01_Schedule.End_Time) ,CONCAT(LN01_Weekly_Schedule.Sunday._1st_Shift_Break1_Start,null,LN01_Schedule._1st_Break_Time) ,CONCAT(LN01_Weekly_Schedule.Sunday._1st_Shift_Lunch_Start,null,LN01_Schedule.Lunch_Time) ,CONCAT(LN01_Weekly_Schedule.Sunday._1st_Shift_Break2_Start,null,LN01_Schedule._2nd_Break_Time) ,MOV(LN01_Weekly_Schedule.Sunday._1st_Shift_Break1_Length,Break1_Length) ,MOV(LN01_Weekly_Schedule.Sunday._1st_Shift_Break2_Length,Break2_Length) ,MOV(LN01_Weekly_Schedule.Sunday._1st_Shift_Lunch_Length,Lunch_Length) ,MOV(LN01_Weekly_Schedule.Sunday.S1_Scheduled,LN01_Schedule.Scheduled_Units) ];
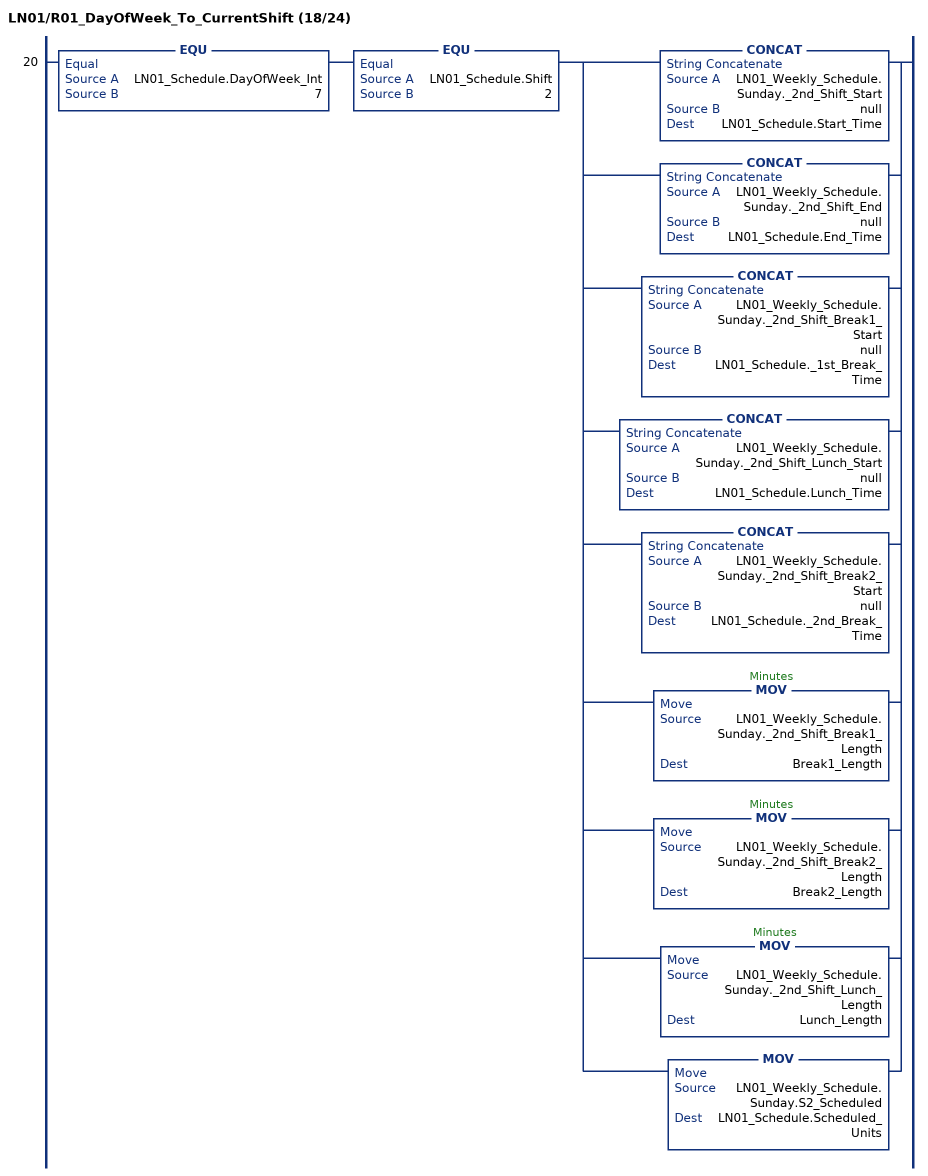
   20: EQU(LN01_Schedule.DayOfWeek_Int,7)EQU(LN01_Schedule.Shift,2)[CONCAT(LN01_Weekly_Schedule.Sunday._2nd_Shift_Start,null,LN01_Schedule.Start_Time) ,CONCAT(LN01_Weekly_Schedule.Sunday._2nd_Shift_End,null,LN01_Schedule.End_Time) ,CONCAT(LN01_Weekly_Schedule.Sunday._2nd_Shift_Break1_Start,null,LN01_Schedule._1st_Break_Time) ,CONCAT(LN01_Weekly_Schedule.Sunday._2nd_Shift_Lunch_Start,null,LN01_Schedule.Lunch_Time) ,CONCAT(LN01_Weekly_Schedule.Sunday._2nd_Shift_Break2_Start,null,LN01_Schedule._2nd_Break_Time) ,MOV(LN01_Weekly_Schedule.Sunday._2nd_Shift_Break1_Length,Break1_Length) ,MOV(LN01_Weekly_Schedule.Sunday._2nd_Shift_Break2_Length,Break2_Length) ,MOV(LN01_Weekly_Schedule.Sunday._2nd_Shift_Lunch_Length,Lunch_Length) ,MOV(LN01_Weekly_Schedule.Sunday.S2_Scheduled,LN01_Schedule.Scheduled_Units) ];
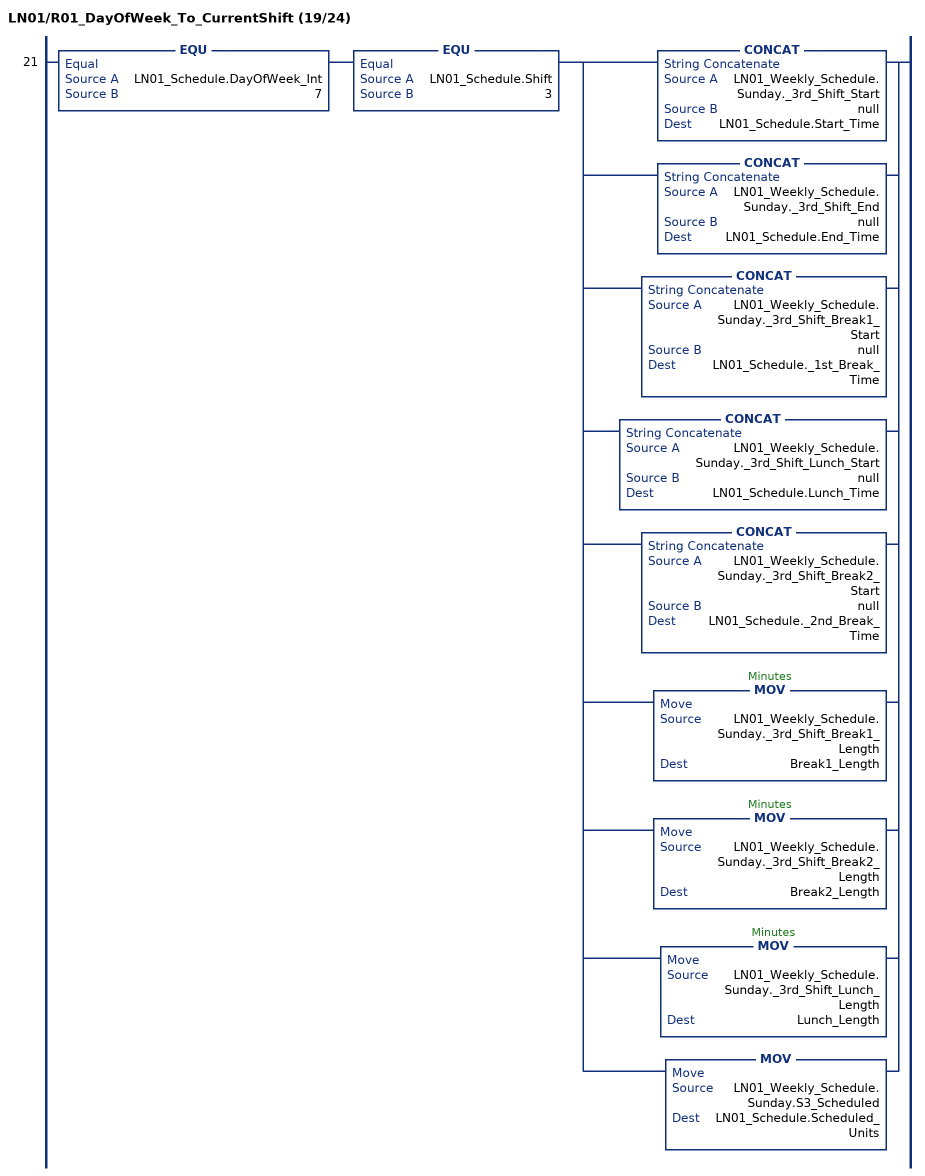
   21: EQU(LN01_Schedule.DayOfWeek_Int,7)EQU(LN01_Schedule.Shift,3)[CONCAT(LN01_Weekly_Schedule.Sunday._3rd_Shift_Start,null,LN01_Schedule.Start_Time) ,CONCAT(LN01_Weekly_Schedule.Sunday._3rd_Shift_End,null,LN01_Schedule.End_Time) ,CONCAT(LN01_Weekly_Schedule.Sunday._3rd_Shift_Break1_Start,null,LN01_Schedule._1st_Break_Time) ,CONCAT(LN01_Weekly_Schedule.Sunday._3rd_Shift_Lunch_Start,null,LN01_Schedule.Lunch_Time) ,CONCAT(LN01_Weekly_Schedule.Sunday._3rd_Shift_Break2_Start,null,LN01_Schedule._2nd_Break_Time) ,MOV(LN01_Weekly_Schedule.Sunday._3rd_Shift_Break1_Length,Break1_Length) ,MOV(LN01_Weekly_Schedule.Sunday._3rd_Shift_Break2_Length,Break2_Length) ,MOV(LN01_Weekly_Schedule.Sunday._3rd_Shift_Lunch_Length,Lunch_Length) ,MOV(LN01_Weekly_Schedule.Sunday.S3_Scheduled,LN01_Schedule.Scheduled_Units) ];
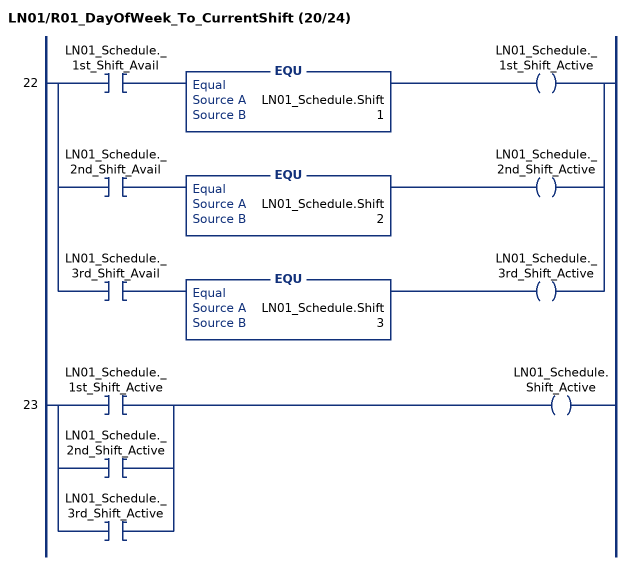
   22: [XIC(LN01_Schedule._1st_Shift_Avail) EQU(LN01_Schedule.Shift,1) OTE(LN01_Schedule._1st_Shift_Active) ,XIC(LN01_Schedule._2nd_Shift_Avail) EQU(LN01_Schedule.Shift,2) OTE(LN01_Schedule._2nd_Shift_Active) ,XIC(LN01_Schedule._3rd_Shift_Avail) EQU(LN01_Schedule.Shift,3) OTE(LN01_Schedule._3rd_Shift_Active) ];
   23: [XIC(LN01_Schedule._1st_Shift_Active) ,XIC(LN01_Schedule._2nd_Shift_Active) ,XIC(LN01_Schedule._3rd_Shift_Active) ]OTE(LN01_Schedule.Shift_Active);
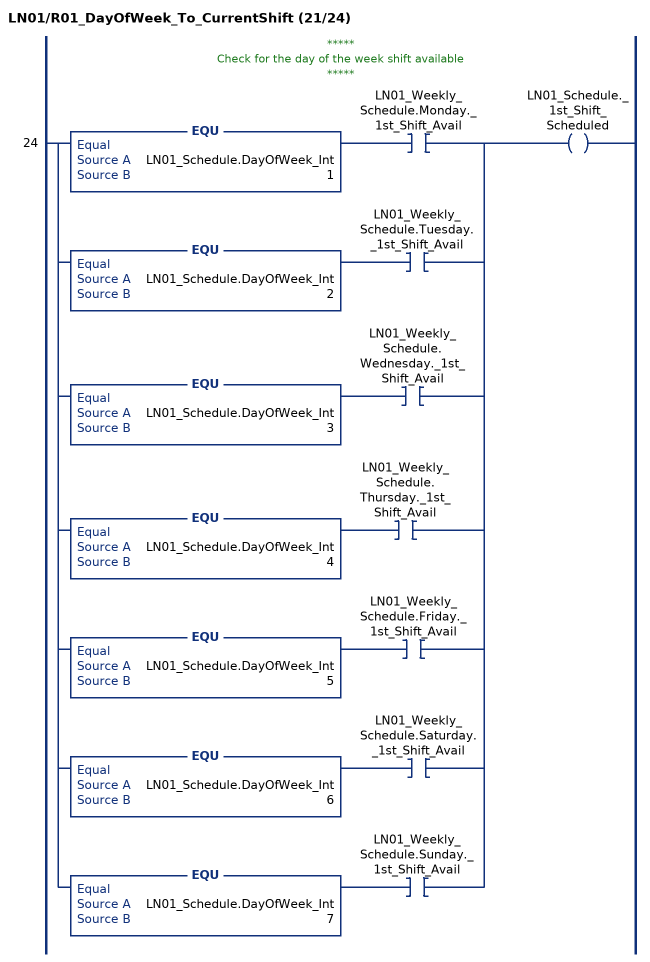
   // *****
   // Check for the day of the week shift available
   // *****
   24: [EQU(LN01_Schedule.DayOfWeek_Int,1) XIC(LN01_Weekly_Schedule.Monday._1st_Shift_Avail) ,EQU(LN01_Schedule.DayOfWeek_Int,2) XIC(LN01_Weekly_Schedule.Tuesday._1st_Shift_Avail) ,EQU(LN01_Schedule.DayOfWeek_Int,3) XIC(LN01_Weekly_Schedule.Wednesday._1st_Shift_Avail) ,EQU(LN01_Schedule.DayOfWeek_Int,4) XIC(LN01_Weekly_Schedule.Thursday._1st_Shift_Avail) ,EQU(LN01_Schedule.DayOfWeek_Int,5) XIC(LN01_Weekly_Schedule.Friday._1st_Shift_Avail) ,EQU(LN01_Schedule.DayOfWeek_Int,6) XIC(LN01_Weekly_Schedule.Saturday._1st_Shift_Avail) ,EQU(LN01_Schedule.DayOfWeek_Int,7) XIC(LN01_Weekly_Schedule.Sunday._1st_Shift_Avail) ]OTE(LN01_Schedule._1st_Shift_Scheduled);
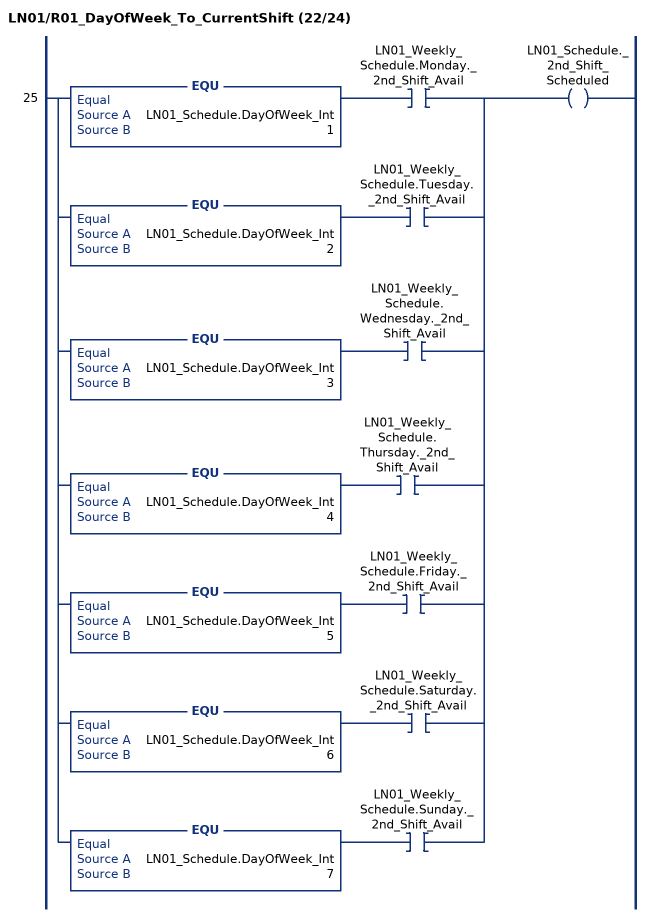
   25: [EQU(LN01_Schedule.DayOfWeek_Int,1) XIC(LN01_Weekly_Schedule.Monday._2nd_Shift_Avail) ,EQU(LN01_Schedule.DayOfWeek_Int,2) XIC(LN01_Weekly_Schedule.Tuesday._2nd_Shift_Avail) ,EQU(LN01_Schedule.DayOfWeek_Int,3) XIC(LN01_Weekly_Schedule.Wednesday._2nd_Shift_Avail) ,EQU(LN01_Schedule.DayOfWeek_Int,4) XIC(LN01_Weekly_Schedule.Thursday._2nd_Shift_Avail) ,EQU(LN01_Schedule.DayOfWeek_Int,5) XIC(LN01_Weekly_Schedule.Friday._2nd_Shift_Avail) ,EQU(LN01_Schedule.DayOfWeek_Int,6) XIC(LN01_Weekly_Schedule.Saturday._2nd_Shift_Avail) ,EQU(LN01_Schedule.DayOfWeek_Int,7) XIC(LN01_Weekly_Schedule.Sunday._2nd_Shift_Avail) ]OTE(LN01_Schedule._2nd_Shift_Scheduled);
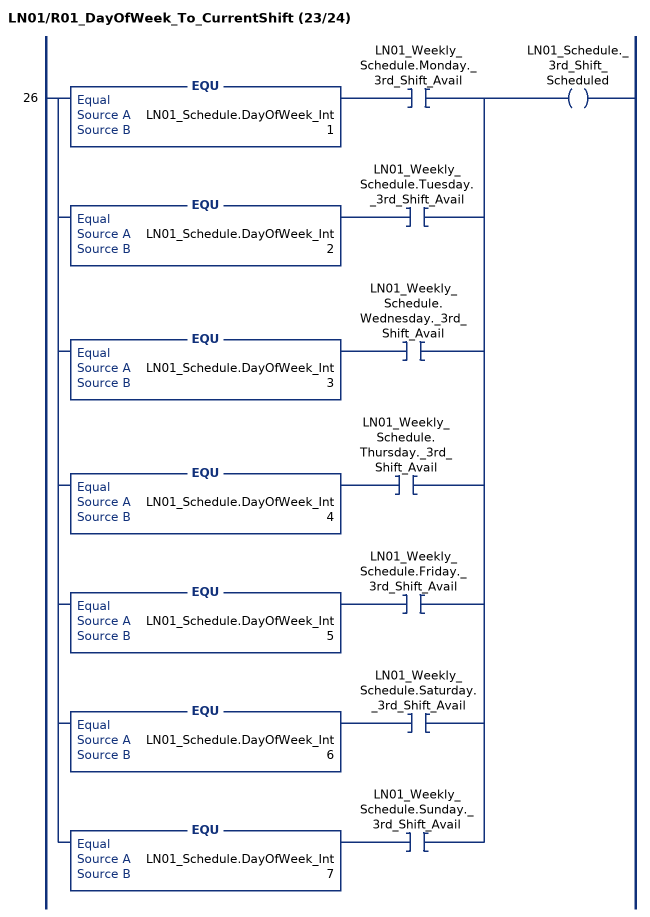
   26: [EQU(LN01_Schedule.DayOfWeek_Int,1) XIC(LN01_Weekly_Schedule.Monday._3rd_Shift_Avail) ,EQU(LN01_Schedule.DayOfWeek_Int,2) XIC(LN01_Weekly_Schedule.Tuesday._3rd_Shift_Avail) ,EQU(LN01_Schedule.DayOfWeek_Int,3) XIC(LN01_Weekly_Schedule.Wednesday._3rd_Shift_Avail) ,EQU(LN01_Schedule.DayOfWeek_Int,4) XIC(LN01_Weekly_Schedule.Thursday._3rd_Shift_Avail) ,EQU(LN01_Schedule.DayOfWeek_Int,5) XIC(LN01_Weekly_Schedule.Friday._3rd_Shift_Avail) ,EQU(LN01_Schedule.DayOfWeek_Int,6) XIC(LN01_Weekly_Schedule.Saturday._3rd_Shift_Avail) ,EQU(LN01_Schedule.DayOfWeek_Int,7) XIC(LN01_Weekly_Schedule.Sunday._3rd_Shift_Avail) ]OTE(LN01_Schedule._3rd_Shift_Scheduled);
